// TIA Portal V20 export
VAR_GLOBAL   // PLC tag table "Default tag table"
   tag AT %I0.0 : Bool;
   tag_1 AT %IW100 : Word;
   tag_2 AT %IB104 : Char;
   tag_3 AT %ID105 : DWord;
   tag_4 AT %ID106 : Real;
   tag_5 AT %I0.5 : Bool;
   tag_6 AT %Q0.0 : Bool;
END_VAR
